Universal Robots PolyScope program: thegreatcorholio.urp

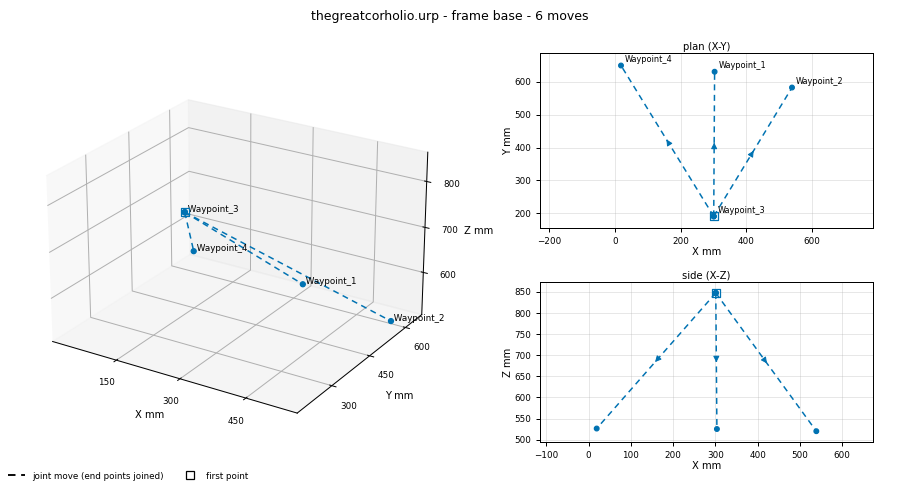
[picture p0: tool path of thegreatcorholio.urp in frame base, 6 of 12 moves have a stored position in this frame; points joined in program order, loops and branches not executed]
Program thegreatcorholio (createdIn=3.4.4.412 lastSavedIn=3.4.4.412 directory=/programs installation=default robotSerialNumber=2017356443)
Calibrated DH parameters: a=[0.000092, -0.116521, -0.182101, -0.000106, 0.000044, 0]; d=[0.089391, 255.189113, -82.629387, -172.449369, 0.094782, 0.082637]; alpha=[1.569598, 0.001603, 0.002015, 1.570234, -1.570307, 0]; deltaTheta=[-0.000017, 1.293309, -0.204843, -1.088417, 0.000036, -0.000078]
Robot Program (runOnlyOnce=false motionType=MoveJ speed=1.047198 acceleration=1.396263 useActiveTCP=false)
